{attribute 'linkalways'} 
{attribute 'no_explicit_call' := 'This FB is a CLASS and must be accessed using methods or properties'}
{attribute 'enable_dynamic_creation'}
FUNCTION_BLOCK Node_RGBA_RANDOM EXTENDS VisionNode
VAR
    out : _TcVnVector4_LREAL;
END_VAR

METHOD PUBLIC  Clone : I_Node
VAR
	pNode : POINTER TO Node_RGBA_RANDOM;
END_VAR
pNode := __NEW(Node_RGBA_RANDOM);
Clone := pNode^;
END_METHOD

METHOD FB_init : BOOL
VAR_INPUT
	bInitRetains : BOOL; // if TRUE, the retain variables are initialized (warm start / cold start)
	bInCopyCode : BOOL;  // if TRUE, the instance afterwards gets moved into the copy code (online change)
END_VAR
AddOutput('out', out);
END_METHOD

METHOD PROTECTED OnExecute
out.Value := GVL_COLOURS.RGBA_RANDOM;
END_METHOD

METHOD PUBLIC PreExecutionCheck
VAR_INPUT
	Check : I_PreExecutionChecks;
END_VAR
END_METHOD

END_FUNCTION_BLOCK

(* stored: Version 1.1.0.1, ProductVersion 3.1.4024.13
   POU Node_RGBA_RANDOM: Id {a4b99d21-1a30-0184-387f-a1e8cdf99d39}, SpecialFunc None
   Folder Constructor: Id {c9789cfa-3dd3-037a-0b6a-69be803ef2b1}
   Method Clone: Id {c825b2c2-12c1-0625-1254-4bfdd7eb2414}
   Method FB_init: Id {ca3905db-9228-0ad9-0bcc-deb12c36ef0a}
   Method OnExecute: Id {f8a37038-213f-09d7-0982-e86500910ae6}
   Method PreExecutionCheck: Id {0b597686-e7de-0a46-20fe-d29ceddaa84d} *)
